Staubli VAL3: matrix.pjx

--- matrix.pjx ---
Parameters version=s8.13.1Cs9_BS2800 stackSize=5000 millimeterUnit=true
Program file=add.pgx
Program file=start.pgx
Program file=stop.pgx
Program file=sub.pgx
Data file=matrix.dtx
Library alias=util path=Disk://helpers/helpers.pjx

--- matrix.dtx ---
mdesc mNomSpeed
num nMatrix1[3 4]
num nMatrix2[3 4]
num nResult[1 1]

--- start.pgx ---
program start()
  local num l_nX
  local num l_nY
begin

  for l_nX = 0 to 2
    for l_nY = 0 to 3
      nMatrix1[l_nX,l_nY] = l_nX*l_nY
      nMatrix2[l_nX,l_nY] = l_nX+l_nY
    endFor
  endFor

  ? "Matrix 1:"
  call util:printNum2d(nMatrix1)
  ? "Matrix 2:"
  call util:printNum2d(nMatrix2)

  ? "test add: add(nMatrix1,nMatrix2, nResult)"
  call add(nMatrix1,nMatrix2, nResult)
  call util:printNum2d(nResult)


end

--- add.pgx ---
public program add(num& x_nMatrix1[] (dimensions=2), num& x_nMatrix2[] (dimensions=2), num& x_nResult[] (dimensions=2))
  local num l_nX
  local num l_nY
begin

  resize(x_nResult,1,size(x_nMatrix1,1))
  resize(x_nResult,2,size(x_nMatrix1,2))

  for l_nX = 0 to size(x_nMatrix1,1)-1
    for l_nY = 0 to size(x_nMatrix1,2)-1
      x_nResult[l_nX,l_nY] = x_nMatrix1[l_nX,l_nY] + x_nMatrix2[l_nX,l_nY]
    endFor
  endFor


end

--- sub.pgx ---
public program sub(num& x_nMatrix1[] (dimensions=2), num& x_nMatrix2[] (dimensions=2), num& x_nResult[] (dimensions=2))
  local num l_nX
  local num l_nY
begin

  resize(x_nResult,1,size(x_nMatrix1,1))
  resize(x_nResult,2,size(x_nMatrix1,2))

  for l_nX = 0 to size(x_nMatrix1,1)-1
    for l_nY = 0 to size(x_nMatrix1,2)-1
      x_nResult[l_nX,l_nY] = x_nMatrix1[l_nX,l_nY] - x_nMatrix2[l_nX,l_nY]
    endFor
  endFor


end
